FUNCTION F_PosUnderUpperBound : BOOL
VAR_INPUT
    fPosition: LREAL;
    stPositionState: DUT_PositionState;
END_VAR

F_PosUnderUpperBound := fPosition < stPositionState.fPosition + ABS(stPositionState.fDelta)

END_FUNCTION

(* stored: Version 1.1.0.1, ProductVersion 3.1.4022.18
   POU F_PosUnderUpperBound: Id {b5ee37fa-13c6-40f2-a7c7-9ac80833d78f}, SpecialFunc None *)
